(*********************************** G.D S.p.A. - Technical Department ***********************************
============= PROGRAM INFO ============
FOLDER:             TBD
MACHINES INVOLVED:  TBD 

============= DESCRIPTION =============
csp machine declaration

============= REVISIONS ===============
Date		Version	 	Author      	Description             
----------	-------		------------  	--------------------------------------------
2019/04/05 	0000.00	 	M.Grasso		Creation of the PRG

**********************************************************************************************************)
(*$R process_ref := prc; $*)
PROGRAM csp_case_topRail_squaring
VAR
	
	prc:											process;
	prc_path:										STRING;
	
END_VAR

_read_var_input();

_object_manager();

IF NOT objects_running()
THEN
	RETURN;	
END_IF

_read_process_image();

_mode_manager();

_set_runtime_properties();

(********************************* BODY *********************************)
(************************************************************************)

_handle_messages();

_write_output();

ACTION _handle_messages:
;
END_ACTION

ACTION _handle_process_test:
;
END_ACTION

ACTION _mode_manager:
IF process_mode_req_is_pending(prc)
THEN
    process_apply_mode_req_first_step(prc);
    CASE process_get_mode(prc) OF
        MODE_TO_ABSENT:
			;
        MODE_TO_INACTIVE:
			;
        MODE_TO_TEST:
			;
        MODE_TO_OPERATIONAL:
			;
    END_CASE
    process_apply_mode_req_second_step(prc);
END_IF
END_ACTION

ACTION _object_manager:
IF objects_initialization()
THEN
	sub_process_init(
		object_name					:= 'csp_case_topRail_squaring.prc', 
		process						:= csp_case_topRail.prc, 
		CONVERSION_this				:= prc);
		
	prc_path 						:= process_get_path(prc);
END_IF

IF objects_running()
THEN
	process_cycle(prc);
END_IF
END_ACTION

ACTION _read_process_image:
;
END_ACTION

ACTION _read_var_input:
;
END_ACTION

ACTION _set_runtime_properties:
;
END_ACTION

ACTION _write_output:
;
END_ACTION

END_PROGRAM

(* stored: Version 1.1.0.1, ProductVersion 3.1.4022.12
   POU csp_case_topRail_squaring: Id {0dccfda7-a898-4256-8ee9-34d34b3acf6f}, SpecialFunc None
   Action _handle_messages: Id {2bf55b53-5289-465f-9d58-2e11bc4b4978}
   Action _handle_process_test: Id {5fb1bba7-7bb4-459e-ac93-8ba34f0e0b22}
   Action _mode_manager: Id {34c68703-5dce-49f5-9d35-246f6f338d87}
   Action _object_manager: Id {b4cee31a-547d-4bf0-9bb8-831742e32a05}
   Action _read_process_image: Id {5cb68d46-3136-455c-bc29-10e75685636f}
   Action _read_var_input: Id {a0f2e97b-b188-470b-b4aa-86d6c9c22778}
   Action _set_runtime_properties: Id {c82c2965-b26c-4ecb-a36b-5d1fdc568ff1}
   Action _write_output: Id {d0fc810b-ba5d-4b8e-ba7c-9698eda5551a} *)
